{attribute 'qualified_only'}
VAR_GLOBAL
	head_roll_right : REAL;
	head_roll_left : REAL;
	
	
END_VAR

(* stored: Version 1.1.0.1, ProductVersion 3.1.4024.4
   GVL data_to_robot: Id {449cc3ce-83c8-40ed-b25c-c6c0939fd523} *)
